(* CODESYS project timer.library
   Company: ESO
   Description: Local Device Control - Timer Library
   Version: 1.0.3.2
   Placeholder: ESO LDC Timer Library
   Author: Mario Kiekebusch
   Title: ESO LDC Timer Library

Project tree, tasks and I/O mapping:
  libraries: ESO MUDPI Library, * (ESO); Tc2_EtherCAT, * (Beckhoff Automation GmbH); Tc2_Standard, * (Beckhoff Automation GmbH); Tc2_System, * (Beckhoff Automation GmbH); Tc2_Utilities, * (Beckhoff Automation GmbH); Tc3_Module, * (Beckhoff Automation GmbH); VisuDialogs, * (System); VisuSymbols, 3.5.10.0 (System)
  DUTs/
    Enumerated/
      data type E_COE_PTP_ADDRESS_TYPE
      data type E_COE_PTP_DELAY_MECHANISM
      data type E_COE_PTP_STATE
      data type E_COE_PTP_TRANSPORT_LAYER
      data type E_COE_PTP_VERSION
      data type E_COE_STATE
      data type E_DIAG_STATE
      data type E_TIME_ERROR
      data type E_TIME_MODE
      data type E_TIME_SIGNAL_QOS
      data type E_TIME_SIGNAL_STATUS
      data type E_TIME_SOURCE
    Structures/
      data type T_COE_PTP_DIAGNOSTICS
      data type T_COE_PTP_ETHERNET
      data type T_COE_PTP_PARAMETERS
      data type T_COE_STAT
      data type T_DIAG_REP_CFG
      data type T_DIAG_REP_STAT
      data type T_IP_ADDRESS
      data type T_PAYLOAD
      data type T_TIME_CFG
      data type T_TIME_INFO
      data type T_TIME_SIGNAL
      data type T_TIME_STAT
  GVLs/
    global variables GVL_TimeConstants
  lib/
  POUs/
    function block FB_ReadEL6688CoE [ST]: DisableCoERead, ExecuteCoERead, FB_init, GetIpaAddr, GetLeapSecond, GetOffsetFromMaster, GetPtpState, IsErrorFree, ReadConfigParameters, ReadEthernetSettings, ReadLeapSecond, ReadOffsetFromMaster, ReadPtpState
    function block FB_SendEL6688Diag [ST]: FB_exit, FB_init, FB_reinit, IpAddressStringToInteger, ReceiveData, SendDiagnosticData, SetConfigurationParameters, TcAddRef, TcQueryInterface, TcRelease
    function block FB_TIME [ST]: CheckNtpSignal, CheckPtpSignal, ComputeNtpOffset, ComputePtpOffset, ComputeSimulationOffset, CycleUpdate, FB_init, GetErrorText, GetMode, GetMudpiTime, GetSource, GetTime, GetUtcTime, MudpiTimeToDc, PublishPtpDiagnostics, RPC_GetMode, RPC_GetUTC, RPC_SetMode, RPC_SetTime, SetDefaultMode, SetMode, SetSource, SetTime
    program MAIN [ST]
  Version/
    global variables Global_Version
  VISUs/
    Templates/
      visualisation GUI_TEMPLATE_TIME
    visualisation GUI_time_info
  text list GlobalTextList
*)

// DUTs/Enumerated/E_COE_PTP_ADDRESS_TYPE
{attribute 'qualified_only'}
{attribute 'strict'}
TYPE E_COE_PTP_ADDRESS_TYPE :
(
	UNKNOWN := -1,
	DHCP := 0,
	FIXED := 1
);
END_TYPE

// DUTs/Enumerated/E_COE_PTP_DELAY_MECHANISM
{attribute 'qualified_only'}
{attribute 'strict'}
TYPE E_COE_PTP_DELAY_MECHANISM :
(
	UNKNOWN := -1,
	DISABLED := 0,
	E2E := 1,
	P2P := 2
);
END_TYPE

// DUTs/Enumerated/E_COE_PTP_STATE
{attribute 'qualified_only'}
{attribute 'strict'}
TYPE E_COE_PTP_STATE :
(   
	UNKNOWN := -1,
	LISTENING := 4,
	SLAVE := 9
);
END_TYPE

// DUTs/Enumerated/E_COE_PTP_TRANSPORT_LAYER
{attribute 'qualified_only'}
{attribute 'strict'}
TYPE E_COE_PTP_TRANSPORT_LAYER :
(
	UNKNOWN := -1,
	PTP_OVER_ETHERNET := 0,
	PTP_OVER_UDP := 1
);
END_TYPE

// DUTs/Enumerated/E_COE_PTP_VERSION
{attribute 'qualified_only'}
{attribute 'strict'}
TYPE E_COE_PTP_VERSION :
(
	UNKONWN := -1,
	PTPv1 := 16,
	PTPv2 := 32
);
END_TYPE

// DUTs/Enumerated/E_COE_STATE
{attribute 'qualified_only'}
{attribute 'strict'}
TYPE E_COE_STATE :
(
	E_COE_UNKNOWN := -1,
	E_COE_NOT_STARTED := 0,	
	E_COE_INIT,
	E_COE_IDLE,
	E_COE_READ,
	E_COE_WAITING,
	E_COE_SLEEPING,
	E_COE_ERROR := 100
	
);
END_TYPE

// DUTs/Enumerated/E_DIAG_STATE
{attribute 'qualified_only'}
{attribute 'strict'}
TYPE E_DIAG_STATE :
(
	E_DIAG_DISABLED := -1,
	E_DIAG_INIT := 0,
	E_DIAG_SENDING,
	E_DIAG_WAITING
);
END_TYPE

// DUTs/Enumerated/E_TIME_ERROR
{attribute 'qualified_only'}
{attribute 'strict'}
TYPE E_TIME_ERROR :
(
	OK := 0,
	NO_SIMULATION_MODE,
	DC2TC_OFFSET_NOT_MAPPED,
	INT_EXT_NOT_MAPPED,
	COE_NOT_VALID,
	PTP_WRONG_STATE,
	PTP_NOT_SYNCHRONIZED,
	NTP_NOT_CONNECTED,
	NTP_NOT_SYNCHRONIZED
);
END_TYPE

// DUTs/Enumerated/E_TIME_MODE
{attribute 'qualified_only'}
{attribute 'strict'}
TYPE E_TIME_MODE :
(
	LOCAL,
    UTC_PTP,
	UTC_NTP,
	UTC,
    SIMULATION
);
END_TYPE

// DUTs/Enumerated/E_TIME_SIGNAL_QOS
{attribute 'qualified_only'}
{attribute 'strict'}
TYPE E_TIME_SIGNAL_QOS :
(
	NOT_VALID := 0,
	NOT_SYNCHRONIZED,
	VALID
);
END_TYPE

// DUTs/Enumerated/E_TIME_SIGNAL_STATUS
{attribute 'qualified_only'}
{attribute 'strict'}
TYPE E_TIME_SIGNAL_STATUS :
(
	CONNECTED := 0,
	NOT_CONNECTED
);
END_TYPE

// DUTs/Enumerated/E_TIME_SOURCE
{attribute 'qualified_only'}
{attribute 'strict'}
TYPE E_TIME_SOURCE :
(
	NONE,
	NTP,
    PTP
);
END_TYPE

// DUTs/Structures/T_COE_PTP_DIAGNOSTICS
TYPE T_COE_PTP_DIAGNOSTICS :
STRUCT
	ptp_state: E_COE_PTP_STATE := E_COE_PTP_STATE.UNKNOWN;
	leap_second: INT := 0;
	offset_from_master: DINT := 0;       // offset from master in ns
	offset_from_master_msec: LREAL := 0;  // offset from master in ms
	offset_from_master_sec: LREAL := 0;   // offset from master in sec
	mean_path_delay: DINT := 0;
END_STRUCT
END_TYPE

// DUTs/Structures/T_COE_PTP_ETHERNET
TYPE T_COE_PTP_ETHERNET :
STRUCT
	address_type: E_COE_PTP_ADDRESS_TYPE := E_COE_PTP_ADDRESS_TYPE.UNKNOWN;
	ip_address_arr:   DWORD;         
	ip_address:       T_IPv4Addr;
	subnet_mask_arr:  DWORD;
	subnet_mask:      T_IPv4Addr;
	gateway_arr:      DWORD;
	gateway:          T_IPv4Addr;
END_STRUCT
END_TYPE

// DUTs/Structures/T_COE_PTP_PARAMETERS
TYPE T_COE_PTP_PARAMETERS :
STRUCT
	ptp_version: E_COE_PTP_VERSION := E_COE_PTP_VERSION.UNKONWN;
	transport_layer: E_COE_PTP_TRANSPORT_LAYER := E_COE_PTP_TRANSPORT_LAYER.UNKNOWN;
	delay_mechanism : E_COE_PTP_DELAY_MECHANISM :=  E_COE_PTP_DELAY_MECHANISM.UNKNOWN;
	ethernet_settings: T_COE_PTP_ETHERNET;	
END_STRUCT
END_TYPE

// DUTs/Structures/T_COE_STAT
TYPE T_COE_STAT :
STRUCT
	diagnostics: T_COE_PTP_DIAGNOSTICS;
	config: T_COE_PTP_PARAMETERS;
	errorFlag: BOOL;
	errorNumber: UDINT;
END_STRUCT
END_TYPE

// DUTs/Structures/T_DIAG_REP_CFG
TYPE T_DIAG_REP_CFG :
STRUCT
	// Configuration parameters related to the TIME diagnostics.
	enabled : BOOL := FALSE; // True if diagnostic data is sent via MUDPI protocol
	address : Tc2_System.T_IPv4Addr := '134.171.2.213'; // Destination IP address for the data
	destination_port: UINT := 7003; // Destination port for the data
	source_port: UINT := 10000;    // Source port of the data
	topic_id: UDINT := 500;      // MUDPI Topic identity
	compontent_id: UINT := 1;  // MUDPI component identity
	sampling: UINT := 10000; // Sampling rate in milliseconds
END_STRUCT
END_TYPE

// DUTs/Structures/T_DIAG_REP_STAT
TYPE T_DIAG_REP_STAT :
STRUCT
	enabled: BOOL; // flag reporting if diagnostic data is being sent externally.
	state : E_DIAG_STATE := E_DIAG_STATE.E_DIAG_DISABLED;
	counter: UDINT; // counter the number of times the diagnostic data was sent.
	last_notification: LREAL; // timestamp of the last sent
	last_notification_date: STRING;
END_STRUCT
END_TYPE

// DUTs/Structures/T_IP_ADDRESS
TYPE T_IP_ADDRESS :
UNION
	ipAdrInternal : UDINT;
	ipAdr : ARRAY[0..3] OF BYTE;
END_UNION
END_TYPE

// DUTs/Structures/T_PAYLOAD
TYPE T_PAYLOAD :
STRUCT
	version:               UINT := 1;
	devtype:               UINT := 10;  // 10: is a Beckhoff PLC according ESO-331947
	hostname:              STRING(16) := '';
    port_state1:	       INT := 0;
	port_state2:           UINT := 0;
	offset_from_master:    LINT := 0;
	mean_path_delay:       ULINT := 0;
	announce_path_delay:   DINT := -1;
	sync_msg_count:        DINT := -1;
	delay_resp_count:      DINT := -1;
	clock_identity:        STRING(8) := '';
	gm_identity:           STRING(8) := '';
	parent_port_identity:  STRING(10) := '';
	current_utc_offset:    INT := 999;
	steps_removed:         UINT := 999;
	error_status:          UINT := 0;
	app_specific:          DINT := 0;
END_STRUCT
END_TYPE

// DUTs/Structures/T_TIME_CFG
TYPE T_TIME_CFG :
STRUCT
	nMode     : E_TIME_MODE := E_TIME_MODE.LOCAL;  // New mode configured.
	nSource   : E_TIME_SOURCE := E_TIME_SOURCE.NONE;  // New mode configured.
	sUserTime : STRING(29) := 'YYYY-MM-DD-hh:mm:ss.nnnnnnnnn'; // Last user configured datetime in format YYYY-MM-DD-hh:mm:ss.nnnnnnnnn
	tUserTime : ULINT := 0;
	nLeapSecond: INT := 37; // Leap second to convert to TAI for systems without PTP.
	
    diag_report: T_DIAG_REP_CFG;	
END_STRUCT
END_TYPE

// DUTs/Structures/T_TIME_INFO
TYPE T_TIME_INFO :
STRUCT
	time_offset :    LINT;
	leap_second:    DINT;  
	time_mode   :    DINT := E_TIME_MODE.LOCAL;
END_STRUCT
END_TYPE

// DUTs/Structures/T_TIME_SIGNAL
TYPE T_TIME_SIGNAL :
STRUCT
	status : E_TIME_SIGNAL_STATUS := E_TIME_SIGNAL_STATUS.NOT_CONNECTED;
	qos    : E_TIME_SIGNAL_QOS    := E_TIME_SIGNAL_QOS.NOT_VALID;
	time_difference : UDINT; // Time difference between DC and External Time Source
	
END_STRUCT
END_TYPE

// DUTs/Structures/T_TIME_STAT
TYPE T_TIME_STAT :
STRUCT
	sLibVersion:	   STRING	:= 'UNKNOWN'; // Library version as string, e.g. '1.2.0.0'
	sSystemTime:       STRING := '';
	sDcTime:           STRING := '';
	sUtcTime:          STRING := '';
	sTaiTime:          STRING := '';
	sErrorMsg:         STRING := '';
	mode:              E_TIME_MODE := E_TIME_MODE.LOCAL;
	source:			   E_TIME_SOURCE := E_TIME_SOURCE.NTP;
	signal:            T_TIME_SIGNAL;
	lNtpOffsetTime:    LINT := 0;
	lPtpOffsetTime:    LINT := 0;
	lSimOffsetTime:    LINT := 0;
	lDcCurrentTime:    LINT := 0;
	lUtcTime:          LINT := 0;   // UTC time in nanoseconds
	lTaiTime:          LINT := 0;   // TAI time in nanoseconds 
	lTaiUnixTime:      LINT := 0;   // UNIX time in nanoseconds
	lrTaiUnixTimeinSecs: LREAL := 0; // UNIX time in seconds - used in MUDPI protocol
	
	sUserTime:         STRING(29) := 'YYYY-MM-DD-hh:mm:ss.nnnnnnnnn'; // Last user configured datetime in format YYYY-MM-DD-hh:mm:ss.nnnnnnnnn
	tUserTime :        ULINT := 0;
	el6688:            T_COE_STAT; 
	diag_report:       T_DIAG_REP_STAT;
	
END_STRUCT
END_TYPE

// GVLs/GVL_TimeConstants
{attribute 'qualified_only'}
VAR_GLOBAL
	C_INVALID:    DINT := -9999;
	C_ONE_SEC:    LINT := 1000000000;
	C_STAT_OK:    DINT := 0;
	C_NS2MSEC:    LREAL := 1/1E+6;
	C_NS2SEC:     LREAL := 1/1E+9;
	C_UNIX_OFFSET_SEC: ULINT := DATE_TO_ULINT(DATE#2000-01-01); // 946,684,800 seconds = 15,778,080 minutes = 262,968 hours
	C_UNIX_OFFSET_MICROSEC:  ULINT := C_UNIX_OFFSET_SEC * 10#1000_000;
END_VAR

// Version/Global_Version
{attribute 'TcGenerated'}
{attribute 'no-analysis'}
{attribute 'linkalways'}
// This function has been automatically generated from the project information.
VAR_GLOBAL CONSTANT
	{attribute 'const_non_replaced'}
	stLibVersion_ESO_LDC_Timer_Library : ST_LibVersion := (iMajor := 1, iMinor := 0, iBuild := 3, iRevision := 2, nFlags := 0, sVersion := '1.0.3.2');
END_VAR

// POUs/FB_ReadEL6688CoE
FUNCTION_BLOCK FB_ReadEL6688CoE
VAR_INPUT
	st_amsAddr:  AMSADDR;
END_VAR
VAR_OUTPUT
END_VAR


VAR_IN_OUT
	i_coe_stat               : T_COE_STAT;
END_VAR

VAR
	  stat: REFERENCE TO T_COE_STAT;
	        
	  fb_SdoLeapSecond   : FB_EcCoESdoRead;
	  fb_SdoPtpState     : FB_EcCoESdoRead;
	  fb_SdoOffset       : FB_EcCoESdoRead;
	  
	  fb_SdoDelayMech    : FB_EcCoESdoRead;
	  fb_SdoPtpVersion   : FB_EcCoESdoRead;
	  fb_SdoTransLayer   : FB_EcCoESdoRead;
	  
	  fb_SdoEtherType    : FB_EcCoESdoRead;
	  fb_SdoEtherIp      : FB_EcCoESdoRead;
	  fb_SdoEtherMask    : FB_EcCoESdoRead;
	  fb_SdoEtherGateway : FB_EcCoESdoRead;
	  
	  
      s_mNetId           : T_AmsNetId;
      b_mCoEExecute      : BOOL;
      n_mSlaveAddr       : UINT;
	  b_CoEReadDiag      : BOOL;    // Flag to trigger reading of diagnostics CoE parameters
	  b_CoEReadCfg       : BOOL;    // Flag to trigger reading of configuration CoE parameters
	  n_state            : E_COE_STATE := E_COE_STATE.E_COE_UNKNOWN;
	  
	  waitTime			 : TIME := T#10000MS;
	  initTime			 : TIME := T#5MS;
	  waitTout			 : TON;    // timer for resting time when reading CoE parameters.
      initTout			 : TON;    // timer for waiting few ms before start reading CoE
END_VAR

stat REF= i_coe_stat; 

CASE n_state OF
	E_COE_STATE.E_COE_NOT_STARTED:
	    initTout (IN := TRUE, PT := initTime); (* enable timer *)
		n_state := E_COE_STATE.E_COE_INIT;
		
	E_COE_STATE.E_COE_INIT:
	    initTout (IN := TRUE);  (* activate timer counting per each cycle *)
		IF initTout.Q THEN
	       n_state := E_COE_STATE.E_COE_IDLE;
		   s_mNetId := F_CreateAmsNetId(st_amsAddr.netId);
		   n_mSlaveAddr := st_amsAddr.port;
		   b_CoEReadCfg := TRUE;
		   b_CoEReadDiag := TRUE;
		   initTout (IN := FALSE);
		END_IF
		
	E_COE_STATE.E_COE_IDLE:
	    waitTout (IN := FALSE); (* Reset timer *)
		DisableCoERead();
	
		 IF (b_CoEReadCfg OR b_CoEReadDiag) THEN
			// Prepare CoE-Access: Read value of CoE object/ sub index
			n_state := E_COE_STATE.E_COE_READ;// Next state for writing
		END_IF
	   
		
	E_COE_STATE.E_COE_READ:
	    waitTout (IN := FALSE); (* Reset timer *)
		stat.errorFlag := FALSE;
	   	stat.errorNumber := 0;
		IF (b_CoEReadCfg) THEN
		 	ReadConfigParameters(st_ioParams := stat.config);	
			b_CoEReadCfg := FALSE;
		END_IF
		IF (b_CoEReadDiag) THEN
	    	ReadLeapSecond(n_iIndex := 16#FA80, 
				n_iSubindex := 11, 
				n_ioLeapSecond := stat.diagnostics.leap_second);
			ReadPtpState(n_iIndex := 16#FA80, 
				n_iSubindex := 2, 
				n_ioPtpState := stat.diagnostics.ptp_state);
	    	ReadOffsetFromMaster(n_iIndex := 16#FA80, 
				n_iSubindex := 6, 
				n_ioOffsetFromMaster := stat.diagnostics.offset_from_master);
			b_CoEReadDiag := FALSE;
		END_IF
				
		n_state := E_COE_STATE.E_COE_WAITING;
		
	E_COE_STATE.E_COE_WAITING:
	    // Execute CoE read until done
				
		ExecuteCoERead(fb_SdoPtpVersion);
		ExecuteCoERead(fb_SdoDelayMech);
		ExecuteCoERead(fb_SdoTransLayer);
	    ExecuteCoERead(fb_SdoEtherType);
		ExecuteCoERead(fb_SdoEtherIp);
		ExecuteCoERead(fb_SdoEtherMask);
		ExecuteCoERead(fb_SdoEtherGateway);
		
	    ExecuteCoERead(fb_SdoLeapSecond);  
		ExecuteCoERead(fb_SdoPtpState);
		ExecuteCoERead(fb_SdoOffset);
			
		IF (NOT fb_SdoEtherType.bBusy) AND
			(NOT fb_SdoEtherIp.bBusy) AND
			(NOT fb_SdoEtherMask.bBusy) AND
			(NOT fb_SdoEtherGateway.bBusy) AND
			(NOT fb_SdoDelayMech.bBusy) AND
			(NOT fb_SdoTransLayer.bBusy) AND
			(NOT fb_SdoPtpVersion.bBusy) AND
			(NOT fb_SdoLeapSecond.bBusy) AND
			(NOT fb_SdoPtpState.bBusy) AND
			(NOT fb_SdoOffset.bBusy) THEN
			    stat.config.ethernet_settings.ip_address := GetIpaAddr(stat.config.ethernet_settings.ip_address_arr);
				stat.config.ethernet_settings.subnet_mask := GetIpaAddr(stat.config.ethernet_settings.subnet_mask_arr);
				stat.config.ethernet_settings.gateway := GetIpaAddr(stat.config.ethernet_settings.gateway_arr);
				stat.diagnostics.offset_from_master_msec := DINT_TO_LREAL(stat.diagnostics.offset_from_master) * GVL_TimeConstants.C_NS2MSEC;
				stat.diagnostics.offset_from_master_sec := DINT_TO_LREAL(stat.diagnostics.offset_from_master) * GVL_TimeConstants.C_NS2SEC;
				n_state := E_COE_STATE.E_COE_SLEEPING;
		END_IF
			
	
		waitTout (IN := TRUE, PT := waitTime); (* enable timer *)
		
	E_COE_STATE.E_COE_SLEEPING:
		DisableCoERead();
	   
		waitTout (IN := TRUE);  (* activate timer counting per each cycle *)
		IF waitTout.Q THEN
	       n_state := E_COE_STATE.E_COE_IDLE;
		   b_CoEReadDiag := TRUE;
		   waitTout (IN := FALSE);
		END_IF
		
	E_COE_STATE.E_COE_ERROR:
       waitTout (IN := FALSE);	
	   waitTout (IN := TRUE, PT := waitTime); (* enable timer *)
	   // TODO: Log the error
	   n_state := E_COE_STATE.E_COE_SLEEPING;
END_CASE

METHOD DisableCoERead
VAR_INPUT
END_VAR

 // CoE configuration parameters
 fb_SdoPtpVersion(bExecute:=FALSE);
 fb_SdoDelayMech(bExecute:=FALSE);
 fb_SdoTransLayer(bExecute:=FALSE);
 fb_SdoEtherType(bExecute:=FALSE);
 fb_SdoEtherIp(bExecute:=FALSE);
 fb_SdoEtherMask(bExecute:=FALSE);
 fb_SdoEtherGateway(bExecute:=FALSE);
	
 // CoE diagnostic parameters
 fb_SdoLeapSecond(bExecute:=FALSE);
 fb_SdoPtpState(bExecute:=FALSE);
 fb_SdoOffset(bExecute:=FALSE);
END_METHOD

METHOD ExecuteCoERead : BOOL

VAR_IN_OUT
	refFb :FB_EcCoESdoRead;
END_VAR

refFb();

IF refFb.bError THEN
	stat.errorFlag := refFb.bError;
	stat.errorNumber := refFb.nErrId;
	n_state := E_COE_STATE.E_COE_ERROR;
END_IF
END_METHOD

METHOD FB_init : BOOL
VAR_INPUT
	bInitRetains : BOOL; // if TRUE, the retain variables are initialized (warm start / cold start)
	bInCopyCode : BOOL;  // if TRUE, the instance afterwards gets moved into the copy code (online change)
END_VAR

initTout (IN := FALSE); (* Reset timer *)
n_state := E_COE_STATE.E_COE_NOT_STARTED;
END_METHOD

METHOD GetIpaAddr : T_IPv4Addr
VAR_INPUT
	in_word : DWORD;
END_VAR

VAR
  ids     : T_IPv4AddrArr := [0, 0, 0, 0];  
  bo_word : DWORD := 0;	
  sIPv4   : T_IPv4Addr := '';
END_VAR

// values in terminal EL6688 have network byte order.
bo_word := BE32_TO_HOST(in_word);

// In order to conver to string using system function, we need an array of bytes.
memcpy(ADR(ids), ADR(bo_word), SIZEOF(bo_word));
	
sIPv4 := F_CreateIPv4Addr( ids );

GetIpaAddr := sIPv4;
RETURN;
END_METHOD

METHOD GetLeapSecond : INT
VAR_INPUT
END_VAR

GetLeapSecond := stat.diagnostics.leap_second;
END_METHOD

METHOD GetOffsetFromMaster : DINT
VAR_INPUT
END_VAR

GetOffsetFromMaster := stat.diagnostics.offset_from_master;
END_METHOD

METHOD GetPtpState : INT
VAR_INPUT
END_VAR
GetPtpState := stat.diagnostics.ptp_state;
END_METHOD

METHOD IsErrorFree : BOOL
VAR_INPUT
END_VAR

IF NOT stat.errorFlag THEN
	IsErrorFree := TRUE;
	return;
END_IF

IsErrorFree := FALSE;
END_METHOD

METHOD ReadConfigParameters 
VAR_INPUT
END_VAR

VAR_IN_OUT
	st_ioParams : T_COE_PTP_PARAMETERS;
END_VAR

fb_SdoPtpVersion(sNetId:= s_mNetId,
    nSlaveAddr := n_mSlaveAddr,
	nIndex := 16#F880, 
	nSubIndex := 1, 
	pDstBuf := ADR(st_ioParams.ptp_version), 
	cbBufLen := SIZEOF(st_ioParams.ptp_version),
	bExecute := TRUE);
	
fb_SdoTransLayer(sNetId:= s_mNetId,
    nSlaveAddr := n_mSlaveAddr,
	nIndex := 16#F882, 
	nSubIndex := 1, 
	pDstBuf := ADR(st_ioParams.transport_layer), 
	cbBufLen := SIZEOF(st_ioParams.transport_layer),
	bExecute := TRUE);
	
 fb_SdoDelayMech(sNetId:= s_mNetId,
    nSlaveAddr := n_mSlaveAddr,
	nIndex := 16#F882, 
	nSubIndex := 5, 
	pDstBuf := ADR(st_ioParams.delay_mechanism), 
	cbBufLen := SIZEOF(st_ioParams.delay_mechanism),
	bExecute := TRUE);

ReadEthernetSettings(n_iIndex := 16#F8E0, 
				st_ioEthernetSettings := st_ioParams.ethernet_settings);
END_METHOD

METHOD ReadEthernetSettings
VAR_INPUT
	n_iIndex     : WORD ;
END_VAR

VAR_IN_OUT
	st_ioEthernetSettings : T_COE_PTP_ETHERNET;
END_VAR

VAR 

END_VAR


fb_SdoEtherType(sNetId:= s_mNetId,
    nSlaveAddr := n_mSlaveAddr,
	nIndex := n_iIndex, 
	nSubIndex := 1, 
	pDstBuf := ADR(st_ioEthernetSettings.address_type), 
	cbBufLen := SIZEOF(st_ioEthernetSettings.address_type),
	bExecute := TRUE);
	
fb_SdoEtherIp(sNetId:= s_mNetId,
    nSlaveAddr := n_mSlaveAddr,
	nIndex := n_iIndex, 
	nSubIndex := 2, 
	pDstBuf := ADR(st_ioEthernetSettings.ip_address_arr), 
	cbBufLen := SIZEOF(st_ioEthernetSettings.ip_address_arr),
	bExecute := TRUE);

	
	
	
fb_SdoEtherMask(sNetId:= s_mNetId,
    nSlaveAddr := n_mSlaveAddr,
	nIndex := n_iIndex, 
	nSubIndex := 3, 
	pDstBuf := ADR(st_ioEthernetSettings.subnet_mask_arr), 
	cbBufLen := SIZEOF(st_ioEthernetSettings.subnet_mask_arr),
	bExecute := TRUE);
	
	
	
fb_SdoEtherGateway(sNetId:= s_mNetId,
    nSlaveAddr := n_mSlaveAddr,
	nIndex := n_iIndex, 
	nSubIndex := 4, 
	pDstBuf := ADR(st_ioEthernetSettings.gateway_arr), 
	cbBufLen := SIZEOF(st_ioEthernetSettings.gateway_arr),
	bExecute := TRUE);
END_METHOD

METHOD ReadLeapSecond : BOOL
VAR_INPUT
	n_iIndex     : WORD ;
	n_iSubindex  : BYTE;
END_VAR

VAR_IN_OUT
	n_ioLeapSecond : INT;
END_VAR
		
//IF (b_CoERead = TRUE) THEN
fb_SdoLeapSecond(sNetId:= s_mNetId,
    nSlaveAddr := n_mSlaveAddr,
	nIndex := n_iIndex, 
	nSubIndex := n_iSubindex, 
	pDstBuf := ADR(n_ioLeapSecond), 
	cbBufLen := SIZEOF(n_ioLeapSecond),
	bExecute := TRUE);
								  
(* Prevent reading more than once the parameter *)			
//b_CoERead := FALSE;
END_METHOD

METHOD ReadOffsetFromMaster : BOOL
VAR_INPUT
	n_iIndex     : WORD ;
	n_iSubindex  : BYTE;
END_VAR

VAR_IN_OUT
	n_ioOffsetFromMaster : DINT;
END_VAR

fb_SdoOffset(sNetId:= s_mNetId,
    nSlaveAddr := n_mSlaveAddr,
	nIndex := n_iIndex, 
	nSubIndex := n_iSubindex, 
	pDstBuf := ADR(n_ioOffsetFromMaster), 
	cbBufLen := SIZEOF(n_ioOffsetFromMaster),
	bExecute := TRUE);
END_METHOD

METHOD ReadPtpState : BOOL
VAR_INPUT
	n_iIndex     : WORD ;
	n_iSubindex  : BYTE;
END_VAR

VAR_IN_OUT
	n_ioPtpState : INT;
END_VAR

fb_SdoPtpState(sNetId:= s_mNetId,
    nSlaveAddr := n_mSlaveAddr,
	nIndex := n_iIndex, 
	nSubIndex := n_iSubindex, 
	pDstBuf := ADR(n_ioPtpState), 
	cbBufLen := SIZEOF(n_ioPtpState),
	bExecute := TRUE);
END_METHOD

END_FUNCTION_BLOCK

// POUs/FB_SendEL6688Diag
(*
    This function blocks aims to pack the EL6688 diagnostic data in MUDPI frames
    and transmit them to Time System using Beckhoffs realtime UDP driver (TF6311). 
    The user of this function blocks needs to do the following in order for the library to work correctly:
    - Initialize the library with configuration parameters
        - Destination IP-address (a multicast address)
        - Destination port
        - Source port
        - Topic identity (see MUDPI-specification)
        - Component identity (see MUDPI-specification)
*)

{attribute 'c++_compatible'}
FUNCTION_BLOCK FB_SendEL6688Diag IMPLEMENTS ITcIoUdpProtocolRecv
VAR_INPUT
END_VAR
VAR_OUTPUT
END_VAR
VAR
	(* TF6311 realtime driver parameters *)
    {attribute 'TcInitSymbol'}
    oid : OTCID;
    ipUdp : ITcIoUdpProtocol;
	nUdpPort : UINT := 10000;
    nReceivedPackets : UINT;
    uLastReceivedIP : T_IP_ADDRESS;
    hrInit : HRESULT;
    hrSend : HRESULT; 
    bSuccessfulInitializationOfRealtimeDriver : BOOL := FALSE; // Indication of whether the realtime driver is properly initialized.

	(* Data/contents parameters *)
    mudpiPacket : ESO_MUDPI.FB_MudpiPacket(topicId := 500, componentId := 10);
    dataToBeSent : ARRAY[0..23] OF BYTE; // 6 parameters, each 4 bytes = 24 bytes
	
	  (* Transmission/communication parameters *)
    _destinationIpAddress : UDINT; // Destination address for the data
    _destinationPort : UINT; // Destination port for the data
    _sourcePort : UINT; // Source port of the data
	
END_VAR

METHOD FB_exit : BOOL
VAR_INPUT
    bInCopyCode : BOOL; // if TRUE, the exit method is called for exiting an instance that is copied afterwards (online change).
END_VAR
IF NOT bInCopyCode THEN // no online change
    IF ipUdp <> 0 THEN
        //ipUdp.UnregisterReceiver(nUdpPort); // Shutdown
        ipUdp.UnregisterReceiver(nUdpPort); // Shutdown
        FW_SafeRelease(ADR(ipUdp));
        FB_exit := TRUE;
    END_IF
END_IF
END_METHOD

METHOD FB_init : BOOL
VAR_INPUT
    bInitRetains : BOOL; // if TRUE, the retain variables are initialized (warm start / cold start)
    bInCopyCode : BOOL;  // if TRUE, the instance afterwards gets moved into the copy code (online change)
END_VAR
MudpiPacket.SetNumFrames(NumFrames := 1);
MudpiPacket.SetFrameId(FrameId := 1);

(*
IF NOT bInCopyCode THEN // no online change
	IF ipUdp = 0 AND oid <> 0 THEN
	    hrInit := FW_ObjMgr_GetObjectInstance(	oid:=oid, 
											iid:=TC_GLOBAL_IID_LIST.IID_ITcIoUdpProtocol, 
											pipUnk:=ADR(ipUdp) );
		IF SUCCEEDED(hrInit) THEN 
			IF  SUCCEEDED(ipUdp.RegisterReceiver(nUdpPort, THIS^)) THEN //open port
				FB_init := TRUE;
			ELSE 
				FB_init := FALSE; 
				FW_SafeRelease(ADR(ipUdp));
			END_IF
		END_IF
	ELSIF oid = 0 THEN 
		FB_init := FALSE; 
		hrInit := ERR_INVALID_PARAM; 				
	END_IF
END_IF
*)
END_METHOD

METHOD FB_reinit : BOOL
IF (ipUdp <> 0) THEN
    //ipUdp.RegisterReceiver(nUdpPort, THIS^);
    ipUdp.RegisterReceiver(nUdpPort, THIS^);
    FB_reinit := TRUE;
END_IF
END_METHOD

METHOD PRIVATE IpAddressStringToInteger : UDINT
VAR_INPUT
    IpAddress : Tc2_System.T_IPv4Addr;
END_VAR
VAR
    IpAddressArray : Tc2_System.T_IPv4AddrArr;
    IpAddressInteger : UDINT;
END_VAR
IpAddressArray := Tc2_System.F_ScanIPv4AddrIds(sIPv4 := IpAddress);
IpAddressInteger := LREAL_TO_UDINT(IpAddressArray[0] * EXPT(256, 3) +
                                   IpAddressArray[1] * EXPT(256, 2) +
                                   IpAddressArray[2] * EXPT(256, 1) +
                                   IpAddressArray[3]);

IpAddressStringToInteger := IpAddressInteger;
END_METHOD

{attribute 'c++_compatible'}
{attribute 'minimal_input_size' := '4'}
{attribute 'pack_mode' := '4'}
{warning 'add method implementation'}
METHOD ReceiveData : HRESULT
VAR_INPUT
	ipAddr	: UDINT;
	udpDestPort	: UINT;
	udpSrcPort	: UINT;
	nData	: UDINT;
	pData	: PVOID;
	pVlan	: POINTER TO ETYPE_VLAN_HEADER := 0;
END_VAR
nReceivedPackets := nReceivedPackets + 1;
uLastReceivedIP.ipAdrInternal := ipAddr;
END_METHOD

(*
    This method carry out the sending of the diagnostic data using the Ethernet network driver.
    The parameters are the array of data to be sent and the timestamp that is required by
	the MUDPI protocol.
*)

METHOD SendDiagnosticData : HRESULT
VAR_INPUT
	payload : POINTER TO T_PAYLOAD; 
	timeStamp : LREAL;
END_VAR
	
VAR
	dataToBeSent : ARRAY[0..87] OF BYTE; 
	
END_VAR


IF ipUdp <> 0 AND bSuccessfulInitializationOfRealtimeDriver = TRUE THEN
	
    // Fill up vector with structure
	memcpy(ADR(dataToBeSent[0]),  ADR(payload^.version), SIZEOF(payload^.version));
	memcpy(ADR(dataToBeSent[2]),  ADR(payload^.devtype), SIZEOF(payload^.devtype));
	memcpy(ADR(dataToBeSent[4]),  ADR(payload^.hostname), SIZEOF(payload^.hostname));
	memcpy(ADR(dataToBeSent[20]), ADR(payload^.port_state1), SIZEOF(payload^.port_state1));
	memcpy(ADR(dataToBeSent[22]), ADR(payload^.port_state2), SIZEOF(payload^.port_state2));
	memcpy(ADR(dataToBeSent[24]), ADR(payload^.offset_from_master), SIZEOF(payload^.offset_from_master));
	memcpy(ADR(dataToBeSent[32]), ADR(payload^.mean_path_delay), SIZEOF(payload^.mean_path_delay));
	memcpy(ADR(dataToBeSent[40]), ADR(payload^.announce_path_delay), SIZEOF(payload^.announce_path_delay));
	memcpy(ADR(dataToBeSent[44]), ADR(payload^.sync_msg_count), SIZEOF(payload^.sync_msg_count));
	memcpy(ADR(dataToBeSent[48]), ADR(payload^.delay_resp_count), SIZEOF(payload^.delay_resp_count));
	memcpy(ADR(dataToBeSent[52]), ADR(payload^.clock_identity), SIZEOF(payload^.clock_identity));
	memcpy(ADR(dataToBeSent[60]), ADR(payload^.gm_identity), SIZEOF(payload^.gm_identity));
	memcpy(ADR(dataToBeSent[68]), ADR(payload^.parent_port_identity), SIZEOF(payload^.parent_port_identity));
	memcpy(ADR(dataToBeSent[78]), ADR(payload^.current_utc_offset), SIZEOF(payload^.current_utc_offset));
	memcpy(ADR(dataToBeSent[80]), ADR(payload^.steps_removed), SIZEOF(payload^.steps_removed));
	memcpy(ADR(dataToBeSent[82]), ADR(payload^.error_status), SIZEOF(payload^.error_status));
	memcpy(ADR(dataToBeSent[84]), ADR(payload^.app_specific), SIZEOF(payload^.app_specific));
	
    // Build MUDPI packet
	mudpiPacket.SetTimeStamp(Timestamp := timeStamp);
    mudpiPacket.SetPayload(payload := ADR(dataToBeSent),
                           payloadSize := SIZEOF(dataToBeSent));
						   
	// Send Data via UDP
    hrSend := ipUdp.SendData(ipDestAddr := _DestinationIpAddress,
                             udpDestPort := _DestinationPort,
                             udpSrcPort := _SourcePort,
                             nData := mudpiPacket.Size(),
                             pData := mudpiPacket.Data(),
                             bCalcUdpCheckSum := FALSE,
                             pVlan := 0);
    IF SUCCEEDED(hrSend) THEN
        mudpiPacket.IncreaseSampleId();
	END_IF
END_IF
END_METHOD

METHOD PUBLIC SetConfigurationParameters
VAR_INPUT
    DestinationIpAddress : Tc2_System.T_IPv4Addr; // Destination IP address for the data
    DestinationPort : UINT; // Destination port for the data
    SourcePort : UINT; // Source port of the data
    TopicId : UDINT; // MUDPI Topic identity
    ComponentId : UINT; // MUDPI component identity
END_VAR
mudpiPacket.SetTopicId(TopicId := TopicId);
mudpiPacket.SetComponentId(ComponentId := ComponentId);

_DestinationIpAddress := IpAddressStringToInteger(IpAddress := DestinationIpAddress);
_DestinationPort := DestinationPort;
_SourcePort := SourcePort;

IF ipUdp = 0 AND NOT bSuccessfulInitializationOfRealtimeDriver THEN
    hrInit := FW_ObjMgr_GetObjectInstance(oid := oid, 
                                          iid := TC_GLOBAL_IID_LIST.IID_ITcIoUdpProtocol,
                                          pipUnk := ADR(ipUdp));
    IF SUCCEEDED(hrInit) THEN
        IF SUCCEEDED(ipUdp.RegisterReceiver(_SourcePort, THIS^)) THEN //open port
            bSuccessfulInitializationOfRealtimeDriver := TRUE;
        ELSE
            FW_SafeRelease(ADR(ipUdp));
        END_IF
    END_IF
END_IF
END_METHOD

{attribute 'c++_compatible'}
{attribute 'minimal_input_size' := '4'}
{attribute 'pack_mode' := '4'}
{warning 'add method implementation'}
METHOD TcAddRef : UDINT
END_METHOD

{attribute 'object_name' := 'TcQueryInterface'}
{attribute 'c++_compatible'}
{attribute 'signature_flag' := '33554688'}
{attribute 'pack_mode' := '4'}
{attribute 'show'}
{attribute 'minimal_input_size' := '4'}
METHOD TcQueryInterface : HRESULT
VAR_INPUT
	iid	: REFERENCE TO IID;
	pipItf	: POINTER TO PVOID;
END_VAR
VAR
	ipUdpRecv : ITcIoUdpProtocolRecv;
	ipUnknown : ITcUnknown;	
END_VAR
IF GuidsEqual(ADR(iid), ADR(TC_GLOBAL_IID_LIST.IID_ITcIoUdpProtocolRecv)) THEN
	ipUdpRecv := THIS^; // cast to interface pointer
	pipItf^ := ITCUNKNOWN_TO_PVOID(ipUdpRecv);
	TcAddRef();
	TcQueryInterface := S_OK;
ELSIF GuidsEqual(ADR(iid), ADR(TC_GLOBAL_IID_LIST.IID_ITcUnknown)) THEN
	ipUnknown := THIS^; // cast to interface pointer
	pipItf^ := ITCUNKNOWN_TO_PVOID(ipUnknown);
	TcAddRef();
	TcQueryInterface := S_OK;
ELSE
	TcQueryInterface := E_HRESULTAdsErr.NOINTERFACE ; //Call super if this fb extends some other
END_IF
END_METHOD

{attribute 'c++_compatible'}
{attribute 'minimal_input_size' := '4'}
{attribute 'pack_mode' := '4'}
{warning 'add method implementation'}
METHOD TcRelease : UDINT
END_METHOD

END_FUNCTION_BLOCK

// POUs/FB_TIME
FUNCTION_BLOCK FB_TIME
VAR_INPUT
END_VAR
VAR_OUTPUT
END_VAR
VAR
	{attribute 'OPC.UA.DA' := '1'}
	{attribute 'OPC.UA.DA.Access' := '1'}
	stat:		T_TIME_STAT;

	{attribute 'OPC.UA.DA' := '1'}
    cfg:         T_TIME_CFG;	
	
	{attribute 'OPC.UA.DA' := '0'}
	fb_CoE:         FB_ReadEL6688CoE;
	
	{attribute 'OPC.UA.DA' := '0'}
	fb_SendDiag:         FB_SendEL6688Diag;
	
	// Input variables from EL6688 
	{attribute 'OPC.UA.DA' := '0'}
	i_inTime               AT %I* : ULINT := 0;
	{attribute 'OPC.UA.DA' := '0'}
	i_exTime               AT %I* : ULINT := 0;
	{attribute 'OPC.UA.DA' := '0'}
	i_dc2TcOffset          AT %I* : LINT := GVL_TimeConstants.C_INVALID;
	{attribute 'OPC.UA.DA' := '0'}
	i_dc2ExtOffset         AT %I* : LINT := GVL_TimeConstants.C_INVALID;
	{attribute 'OPC.UA.DA' := '0'}
	i_extDevNotConnected   AT %I* : BOOL := TRUE;
	{attribute 'OPC.UA.DA' := '0'}
	i_syncMode             AT %I* : UINT;
	{attribute 'OPC.UA.DA' := '0'}
	i_AdsAddr	           AT %I*:	AMSADDR;				// ADS address structure
	{attribute 'OPC.UA.DA' := '0'}
	
	// Input variables from NTP
	{attribute 'OPC.UA.DA' := '0'}
    i_exNtpExtTime               AT %I* : LINT := 0;
	
	{attribute 'OPC.UA.DA' := '0'}
    i_exNtpSysTime         AT %I* : LINT := 0;
	
	{attribute 'OPC.UA.DA' := '0'}
    i_exNtpExtOffset         AT %I* : LINT := 0;
	
	{attribute 'OPC.UA.DA' := '0'}
	i_exNtpConnected   AT %I* : BOOL := FALSE;
	
	{attribute 'OPC.UA.DA' := '0'}
	i_exNtpSynchronized  AT %I* : BOOL := FALSE;
	
	
 	{attribute 'OPC.UA.DA' := '0'}
	q_timeInfo             AT %Q*: T_TIME_INFO;    
	
	rtrigEnableDiagReport        : R_TRIG;
    ftrigDisableDiagReport       : F_TRIG;  
	waitTime			 : TIME := T#10000MS;
	waitTout			 : TON;    // timer for resting time when reading CoE parameters.
	payload              : T_PAYLOAD;
	   
	
END_VAR


fb_CoE(st_amsAddr := i_AdsAddr, i_coe_stat := stat.el6688);
fb_SendDiag();

CycleUpdate();

// If TIMER is configured to send diagnostic reports to the Time System then
// it enables the sending of the data.
rtrigEnableDiagReport(CLK := cfg.diag_report.enabled);
ftrigDisableDiagReport(CLK := cfg.diag_report.enabled);

// Check for the rising edge of the enable flag
IF rtrigEnableDiagReport.Q THEN
	stat.diag_report.state := E_DIAG_STATE.E_DIAG_INIT;
	stat.diag_report.enabled := TRUE;
END_IF

// Check for the falling edge of the enable flag
IF ftrigDisableDiagReport.Q THEN
	stat.diag_report.state := E_DIAG_STATE.E_DIAG_DISABLED;
	stat.diag_report.counter := 0;
	stat.diag_report.enabled := FALSE;
END_IF

CASE stat.diag_report.state OF
E_DIAG_STATE.E_DIAG_INIT:

	fb_SendDiag.SetConfigurationParameters(DestinationIpAddress := cfg.diag_report.address,
		DestinationPort := cfg.diag_report.destination_port,
		SourcePort := cfg.diag_report.source_port,
		TopicId := cfg.diag_report.topic_id,
		ComponentId := cfg.diag_report.compontent_id);
	
	IF DINT_TO_TIME(cfg.diag_report.sampling) < T#500MS THEN
		waitTime := T#500MS;
	ELSE
		waitTime :=  DINT_TO_TIME(cfg.diag_report.sampling);
	END_IF	
	waitTout (IN := TRUE, PT := waitTime); (* enable timer *)
	
	stat.diag_report.state := E_DIAG_STATE.E_DIAG_WAITING;
E_DIAG_STATE.E_DIAG_WAITING:	
	waitTout (IN := TRUE);  (* activate timer counting per each cycle *)
 	IF waitTout.Q THEN
		waitTout (IN := FALSE);
		stat.diag_report.state := E_DIAG_STATE.E_DIAG_SENDING;
 	END_IF
E_DIAG_STATE.E_DIAG_SENDING:  
	// Added information to the payload structure
	// Not all fields are currently supported.
 	payload.port_state1 := fb_CoE.GetPtpState();
	payload.offset_from_master := fb_CoE.GetOffsetFromMaster();
	payload.current_utc_offset := fb_CoE.GetLeapSecond();
	
    fb_SendDiag.SendDiagnosticData(payload := ADR(payload),
					timeStamp := stat.lrTaiUnixTimeinSecs) ;	
	stat.diag_report.counter := stat.diag_report.counter + 1;
	// Reset timer
	waitTout (IN := FALSE);  
	// Go back to the init
	stat.diag_report.state := E_DIAG_STATE.E_DIAG_INIT;
END_CASE

METHOD CheckNtpSignal : BOOL
VAR_INPUT
END_VAR
stat.signal.status :=  E_TIME_SIGNAL_STATUS.CONNECTED;
stat.signal.qos := E_TIME_SIGNAL_QOS.VALID;


// Check external signal. This variable must be mapped to the EL6688 terminal.
IF (NOT i_exNtpConnected) THEN
	stat.signal.status :=  E_TIME_SIGNAL_STATUS.NOT_CONNECTED;
	stat.signal.qos := E_TIME_SIGNAL_QOS.NOT_VALID;
	CheckNtpSignal:=FALSE;
	RETURN;
END_IF	

// Check NTP is synchronized
IF (NOT i_exNtpSynchronized) THEN
	stat.signal.qos := E_TIME_SIGNAL_QOS.NOT_VALID;
	stat.sErrorMsg := GetErrorText(E_TIME_ERROR.NTP_NOT_SYNCHRONIZED);
END_IF	

// Check time delivered by NTP is not zero. This variable
// shall be mapped to the TcNtpExternalTimeProvider
IF (i_exNtpExtTime = 0) THEN
	stat.signal.qos := E_TIME_SIGNAL_QOS.NOT_VALID;
	stat.sErrorMsg := GetErrorText(E_TIME_ERROR.INT_EXT_NOT_MAPPED);
	CheckNtpSignal:=FALSE;
	RETURN;
END_IF


CheckNtpSignal := TRUE;
END_METHOD

METHOD CheckPtpSignal : BOOL
VAR_INPUT
END_VAR
stat.signal.status :=  E_TIME_SIGNAL_STATUS.CONNECTED;
stat.signal.qos := E_TIME_SIGNAL_QOS.VALID;


// Check external signal. This variable must be mapped to the EL6688 terminal.
IF (i_extDevNotConnected) THEN
	stat.signal.status :=  E_TIME_SIGNAL_STATUS.NOT_CONNECTED;
	stat.signal.qos := E_TIME_SIGNAL_QOS.NOT_VALID;
	CheckPtpSignal:=FALSE;
	RETURN;
END_IF	

// Check DC times computed by EL6688 are not zero. These variables
// shall be mapped to the EL6688 terminal.	
IF ((i_inTime = 0) OR (i_exTime = 0)) THEN
	stat.signal.qos := E_TIME_SIGNAL_QOS.NOT_VALID;
	stat.sErrorMsg := GetErrorText(E_TIME_ERROR.INT_EXT_NOT_MAPPED);
	CheckPtpSignal:=FALSE;
	RETURN;
END_IF

IF (i_dc2TcOffset = GVL_TimeConstants.C_INVALID)  THEN
	stat.signal.qos := E_TIME_SIGNAL_QOS.NOT_VALID;
	stat.sErrorMsg := GetErrorText(E_TIME_ERROR.DC2TC_OFFSET_NOT_MAPPED);
	CheckPtpSignal:=FALSE;
	RETURN;
END_IF
		
// Check quality of the signal synchronization. If the offset from master is
// greater than one second if it is consider not synchronized.
IF (ABS(fb_CoE.GetOffsetFromMaster()) >= GVL_TimeConstants.C_ONE_SEC) THEN
	stat.signal.qos := E_TIME_SIGNAL_QOS.NOT_SYNCHRONIZED;
	stat.sErrorMsg := GetErrorText(E_TIME_ERROR.PTP_NOT_SYNCHRONIZED);
END_IF

// Check CoE diagnostic parameter from EL6688. Terminal shall be
// in SLAVE state and not LISTENNING.

IF (NOT fb_CoE.IsErrorFree()) THEN
	stat.signal.qos := E_TIME_SIGNAL_QOS.NOT_VALID;
	stat.sErrorMsg := GetErrorText(E_TIME_ERROR.COE_NOT_VALID);
	CheckPtpSignal:=FALSE;
	RETURN;
END_IF
	
IF (fb_CoE.GetPtpState() <> E_COE_PTP_STATE.SLAVE) THEN
	stat.signal.status :=  E_TIME_SIGNAL_STATUS.NOT_CONNECTED;
	stat.signal.qos := E_TIME_SIGNAL_QOS.NOT_VALID;
	stat.sErrorMsg := GetErrorText(E_TIME_ERROR.PTP_WRONG_STATE);
	CheckPtpSignal:=FALSE;
	RETURN;
END_IF

CheckPtpSignal := TRUE;
END_METHOD

METHOD ComputeNtpOffset
VAR_INPUT
END_VAR

VAR
	dcExtNtpTime : LINT;
	dcExtNtpLocalTime : LINT;
	tmp : ULINT;
	nFileTime : T_FILETIME;
	str: STRING;
END_VAR



MEMCPY(ADR(nFileTime), ADR(i_exNtpExtTime), SIZEOF(nFileTime));

dcExtNtpTime := FILETIME_TO_DCTIME64(nFileTime);
MEMCPY(ADR(nFileTime), ADR(i_exNtpSysTime), SIZEOF(nFileTime));
dcExtNtpLocalTime := FILETIME_TO_DCTIME64(nFileTime);
stat.lNtpOffsetTime := dcExtNtpLocalTime - dcExtNtpTime;

stat.lTaiTime := stat.lDcCurrentTime - stat.lNtpOffsetTime + (UINT_TO_LINT(cfg.nLeapSecond) * GVL_TimeConstants.C_ONE_SEC);
stat.sTaiTime := DCTIME64_TO_STRING(LINT_TO_ULINT(stat.lTaiTime));

// Convert TAI time from nanoseconds to microseconds
tmp := LINT_TO_ULINT(stat.lTaiTime)/ 10#1000;

// Add offset wrt Unix Base System
tmp := tmp + GVL_TimeConstants.C_UNIX_OFFSET_MICROSEC;

// Convert offset from microseconds to seconds for the MUDPI protocol
stat.lrTaiUnixTimeinSecs := ULINT_TO_LREAL(tmp) / 1000000.0;


stat.lUtcTime := stat.lDcCurrentTime - stat.lNtpOffsetTime;						
stat.sUtcTime := DCTIME64_TO_STRING(LINT_TO_ULINT(stat.lUtcTime));
q_timeInfo.time_offset := stat.lNtpOffsetTime;
q_timeInfo.leap_second := cfg.nLeapSecond;
END_METHOD

METHOD ComputePtpOffset
VAR_INPUT
END_VAR

VAR
	dc2ExtOffset : LINT;
	taiOffset : LINT;
	tmp : LREAL;
END_VAR

dc2ExtOffset := ULINT_TO_LINT(i_inTime) - ULINT_TO_LINT(i_exTime);

taiOffset := dc2ExtOffset + i_dc2TcOffset;

stat.lPtpOffsetTime := (dc2ExtOffset) + i_dc2TcOffset +
                           (GVL_TimeConstants.C_ONE_SEC *  fb_CoE.GetLeapSecond());

stat.lTaiTime := stat.lDcCurrentTime - taiOffset;
stat.sTaiTime := DCTIME64_TO_STRING(LINT_TO_ULINT(stat.lTaiTime));

// Convert TAI time from nanoseconds to microseconds
tmp := LINT_TO_REAL(stat.lTaiTime)/ 10#1000;

// Add offset wrt Unix Base System
tmp := tmp + ULINT_TO_REAL(GVL_TimeConstants.C_UNIX_OFFSET_MICROSEC);

// Convert offset from microseconds to seconds for the MUDPI protocol
stat.lrTaiUnixTimeinSecs := tmp / 1000000.0;

stat.lUtcTime := stat.lDcCurrentTime - stat.lPtpOffsetTime;							
stat.sUtcTime := DCTIME64_TO_STRING(LINT_TO_ULINT(stat.lUtcTime));
q_timeInfo.time_offset := stat.lPtpOffsetTime;
q_timeInfo.leap_second := fb_CoE.GetLeapSecond();
END_METHOD

METHOD ComputeSimulationOffset
VAR_INPUT
END_VAR

VAR
	lSimOffsetTime:	LINT	:= 0;
	tDcUserTime      : ULINT;
	tmp : ULINT;
END_VAR

// Get the time from the user given time string, e.g.
// cfg.sUserTime = '2019-12-07-07:07:07.380500000'
// tDcUserTime   = 629017627380500000
tDcUserTime  := STRING_TO_DCTIME64(cfg.sUserTime);
// Adjust the offset only if user modified the time string.
IF (stat.tUserTime <> tDcUserTime) THEN
	IF (tDcUserTime = 0) THEN
		stat.sErrorMsg := 'ERROR: format of user datetime is not correct';
		RETURN;
	END_IF
	lSimOffsetTime := (stat.lDcCurrentTime - ULINT_TO_LINT(tDcUserTime));
	stat.lSimOffsetTime := lSimOffsetTime;
	stat.tUserTime := tDcUserTime;
END_IF

stat.lUtcTime := stat.lDcCurrentTime - stat.lSimOffsetTime;
stat.sUtcTime := DCTIME64_TO_STRING(LINT_TO_ULINT(stat.lUtcTime));
stat.lTaiTime := stat.lUtcTime + (GVL_TimeConstants.C_ONE_SEC * cfg.nLeapSecond);
stat.sTaiTime := DCTIME64_TO_STRING(LINT_TO_ULINT(stat.lTaiTime));;
// Convert TAI time from nanoseconds to microseconds
tmp := LINT_TO_ULINT(stat.lTaiTime)/ 10#1000;

// Add offset wrt Unix Base System
tmp := tmp + GVL_TimeConstants.C_UNIX_OFFSET_MICROSEC;

// Convert offset from microseconds to seconds for the MUDPI protocol
stat.lrTaiUnixTimeinSecs := ULINT_TO_LREAL(tmp) / 1000000.0;
q_timeInfo.time_offset := stat.lSimOffsetTime;
q_timeInfo.leap_second := cfg.nLeapSecond;
END_METHOD

METHOD CycleUpdate : BOOL
VAR_INPUT
END_VAR
VAR
	fbGetSystemTime  : GETSYSTEMTIME;
    fileTime         : T_FILETIME;
	tDcCurrentTime	 : LINT;
	tDcUserTime      : ULINT;
    sTime            : STRING;
	bSignalOk        : BOOL := FALSE;
END_VAR
VAR_INST
	{attribute 'OPC.UA.DA' := '0'}
	lSimOffsetTime:	LINT	:= 0;
END_VAR
// Get System Time
fbGetSystemTime(timeLoDW=>fileTime.dwLowDateTime, timeHiDW=>fileTime.dwHighDateTime );
stat.sSystemTime := SYSTEMTIME_TO_STRING( FILETIME_TO_SYSTEMTIME( fileTime ) );

// Get DC Time
tDcCurrentTime	:= ULINT_TO_LINT(F_GetCurDcTaskTime64());
stat.lDcCurrentTime := tDcCurrentTime; 
stat.sDcTime := DCTIME64_TO_STRING(LINT_TO_ULINT(tDcCurrentTime));	(* DC time as STRING *)


IF (cfg.nMode =  E_TIME_MODE.LOCAL) THEN
	// In local mode, time used is the time DC time delivered by TwinCAT.
	SetDefaultMode('');
ELSIF (cfg.nMode =  E_TIME_MODE.UTC_PTP)  THEN
	stat.sErrorMsg := '';
	// Check PTP time signal.
	// This will set:
	//	stat.signal.status
	//	stat.signal.qos
	bSignalOk := CheckPtpSignal();
	IF bSignalOk	THEN
		stat.mode := E_TIME_MODE.UTC_PTP;
		ComputePtpOffset();	
	ELSE
		SetDefaultMode('PTP signal NOT ok');
	END_IF
ELSIF (cfg.nMode =  E_TIME_MODE.UTC_NTP)  THEN
	stat.sErrorMsg := '';
	// Check NTP time signal.
	// This will set:
	//	stat.signal.status
	//	stat.signal.qos
	bSignalOk := CheckNtpSignal();
	IF bSignalOk	THEN
		stat.mode := E_TIME_MODE.UTC_NTP;
		// This call computes:
		//	stat.lUtcTime							
		//	stat.sUtcTime
		//	q_timeInfo.time_offset
		ComputeNtpOffset();	
	ELSE
		SetDefaultMode(GetErrorText(E_TIME_ERROR.NTP_NOT_CONNECTED));
	END_IF
ELSIF  (cfg.nMode =  E_TIME_MODE.SIMULATION ) THEN
	// Uses the simulated time
	stat.mode := E_TIME_MODE.SIMULATION;
	stat.sErrorMsg := '';
	// This call computes:
			//	stat.tUserTime							
			//	stat.sUtcTime
			//	q_timeInfo.time_offset
	ComputeSimulationOffset();	
END_IF

q_timeInfo.time_mode := stat.mode;
END_METHOD

METHOD FB_init : BOOL
VAR_INPUT
	bInitRetains : BOOL; // if TRUE, the retain variables are initialized (warm start / cold start)
	bInCopyCode : BOOL;  // if TRUE, the instance afterwards gets moved into the copy code (online change)
END_VAR
stat.sLibVersion := stLibVersion_ESO_LDC_Timer_Library.sVersion;
stat.sErrorMsg := '';
END_METHOD

METHOD GetErrorText : STRING
VAR_INPUT
	i_errorId: DINT;
END_VAR

VAR
	str:	STRING;
END_VAR

CASE i_errorId OF
	E_TIME_ERROR.OK:						str	:= 'OK';
	E_TIME_ERROR.NO_SIMULATION_MODE:	    str	:= 'ERROR: Time can only be set in simulation mode.';	
	E_TIME_ERROR.INT_EXT_NOT_MAPPED:        str := 'ERROR: Did you forget to map the internal or external EL6688 time stamps?';
	E_TIME_ERROR.DC2TC_OFFSET_NOT_MAPPED:   str := 'ERROR: Did you forget to map the dc2tc_offset?';
	E_TIME_ERROR.COE_NOT_VALID:             str := 'ERROR: Error reading COE parameter';
	E_TIME_ERROR.PTP_WRONG_STATE:           str := 'ERROR: EL6688 is not in SLAVE state';
	E_TIME_ERROR.NTP_NOT_CONNECTED:         str := 'ERROR: NTP not connected. Did you forget to map attributes?';
	E_TIME_ERROR.NTP_NOT_SYNCHRONIZED:      str := 'WARNING: NTP not synchronized';
END_CASE

GetErrorText	:= str;
END_METHOD

METHOD GetMode : E_TIME_MODE
VAR_INPUT
END_VAR
GetMode := stat.mode;
END_METHOD

METHOD GetMudpiTime : LREAL
VAR_INPUT
END_VAR

VAR
END_VAR

GetMudpiTime := stat.lrTaiUnixTimeinSecs;
END_METHOD

METHOD GetSource : E_TIME_SOURCE
VAR_INPUT
END_VAR
GetSource := stat.source;
END_METHOD

METHOD GetTime : ULINT
VAR_INPUT
END_VAR

IF (GetMode() =  E_TIME_MODE.LOCAL) THEN
	GetTime := LINT_TO_ULINT(stat.lDcCurrentTime);
END_IF

IF (GetMode() =  E_TIME_MODE.UTC_PTP) THEN
	GetTime := LINT_TO_ULINT(stat.lDcCurrentTime - stat.lPtpOffsetTime);
END_IF

IF (GetMode() =  E_TIME_MODE.UTC_NTP) THEN
	GetTime := LINT_TO_ULINT(stat.lDcCurrentTime - stat.lNtpOffsetTime);
END_IF

IF (GetMode() =  E_TIME_MODE.SIMULATION) THEN
	GetTime := LINT_TO_ULINT(stat.lDcCurrentTime - stat.lPtpOffsetTime);
END_IF
END_METHOD

METHOD GetUtcTime : ULINT
VAR_INPUT
END_VAR

VAR
END_VAR

GetUtcTime := i_exNtpSysTime;
END_METHOD

METHOD MudpiTimeToDc : ULINT
VAR_INPUT
	mudipiTime: LREAL;
END_VAR

VAR
	tmp: LREAL;
END_VAR

// Convert offset from seconds (MUDPI protocol) to microseconds 
tmp := mudipiTime * 1000000.0;

// Remove offset wrt Unix Base System
tmp := tmp - ULINT_TO_LREAL(GVL_TimeConstants.C_UNIX_OFFSET_MICROSEC);

// Convert offset from microseconds to nanoseconds - DC unit
tmp := tmp * 10#1000;

MudpiTimeToDc := LREAL_TO_ULINT(tmp);
END_METHOD

(*
  This method sends the diagnostic data to the TRS system for long term
  monitoring.
  
  The format of the data follows the specification in document ESO-331947.
  The data is sent via UDP packets using the implementation of the MUDPI
  protocol.
  *)

METHOD PublishPtpDiagnostics : BOOL
VAR_INPUT
END_VAR

VAR
    (* TF6311 realtime driver parameters *)
    {attribute 'TcInitSymbol'}
    oid : OTCID;
    ipUdp : ITcIoUdpProtocol;
    nReceivedPackets : UINT;
    uLastReceivedIP : T_IP_ADDRESS;
    hrInit : HRESULT;
    hrSend : HRESULT; 
    bSuccessfulInitializationOfRealtimeDriver : BOOL := FALSE; // Indication of whether the realtime driver is properly initialized.

    (* Data/contents parameters *)
    MudpiPacket : ESO_MUDPI.FB_MudpiPacket(topicId := 500, componentId := 10);

    (* Transmission/communication parameters *)
    _DestinationIpAddress : UDINT; // Destination address for the data
    _DestinationPort : UINT; // Destination port for the data
    _SourcePort : UINT; // Source port of the data

   
END_VAR
END_METHOD

{attribute 'TcRpcEnable':='1'}
METHOD RPC_GetMode : E_TIME_MODE
VAR_INPUT
END_VAR

RPC_GetMode := GetMode();
END_METHOD

{attribute 'TcRpcEnable':='1'}
METHOD RPC_GetUTC : STRING(255)
VAR_INPUT
END_VAR

VAR
	part1: STRING;
	part2: STRING;
	timeStr: STRING(255);
END_VAR

CASE stat.mode OF
	E_TIME_MODE.LOCAL:
		part2 := ' Mode: LOCAL';
	E_TIME_MODE.UTC:
	    part2 := ' Mode: UTC';
	E_TIME_MODE.SIMULATION:
	    part2 := ' Mode: SIMULATION';
END_CASE

part1 := CONCAT('UTC: ', stat.sUtcTime);
timeStr := CONCAT(part1, part2);
RPC_GetUTC := timeStr;
END_METHOD

{attribute 'TcRpcEnable':='1'}
METHOD RPC_SetMode : DINT
VAR_INPUT
	in_mode : E_TIME_MODE;
END_VAR

RPC_SetMode := SetMode(in_mode);
END_METHOD

{attribute 'TcRpcEnable':='1'}
METHOD RPC_SetTime : DINT

VAR_INPUT
	in_time : STRING(29);
END_VAR

RPC_SetTime := SetTime(in_time);
END_METHOD

METHOD SetDefaultMode
VAR_INPUT
	str: STRING := '';
END_VAR

VAR
	tmp : ULINT;
END_VAR
// Time signal not OK. Go to LOCAL mode.
cfg.nMode := E_TIME_MODE.LOCAL;
cfg.nSource := E_TIME_SOURCE.NONE;
stat.mode := E_TIME_MODE.LOCAL;
stat.signal.qos := E_TIME_SIGNAL_QOS.NOT_VALID;
stat.lUtcTime := stat.lDcCurrentTime;
stat.sUtcTime := stat.sDcTime;
IF (str <> '') THEN
	stat.sErrorMsg := str;
END_IF
stat.lTaiTime := stat.lDcCurrentTime;
stat.sTaiTime := stat.sDcTime;
//stat.lSimOffsetTime := 0;  

// Convert TAI time from nanoseconds to microseconds
tmp := LINT_TO_ULINT(stat.lTaiTime)/ 10#1000;
// Add offset wrt Unix Base System
tmp := tmp + GVL_TimeConstants.C_UNIX_OFFSET_MICROSEC;
// Convert offset from microseconds to seconds for the MUDPI protocol
stat.lrTaiUnixTimeinSecs := ULINT_TO_LREAL(tmp) / 1000000.0;				

q_timeInfo.time_offset := 0;
q_timeInfo.leap_second := 0;
END_METHOD

METHOD SetMode : DINT
VAR_INPUT
	i_mode : E_TIME_MODE;
END_VAR

cfg.nMode := i_mode;

SetMode := GVL_TimeConstants.C_STAT_OK;
END_METHOD

METHOD SetSource : DINT
VAR_INPUT
	i_source : E_TIME_SOURCE;
END_VAR

cfg.nSource := i_source;

SetSource := GVL_TimeConstants.C_STAT_OK;
END_METHOD

METHOD SetTime : DINT;

VAR_INPUT
	in_time : STRING(29);
END_VAR

VAR
	dc_time :ULINT;
END_VAR

IF (cfg.nMode <> E_TIME_MODE.SIMULATION) THEN
	stat.sErrorMsg := GetErrorText(E_TIME_ERROR.NO_SIMULATION_MODE); 
	SetTime := E_TIME_ERROR.NO_SIMULATION_MODE;
	RETURN;
END_IF

cfg.sUserTime := in_time;
dc_time := STRING_TO_DCTIME64(in_time);
cfg.tUserTime := dc_time;
//st_stat.lSimOffsetTime := (st_stat.lDcCurrentTime - ULINT_TO_LINT(dc_time));
//q_timeInfo.time_offset := st_stat.lSimOffsetTime;
SetTime := GVL_TimeConstants.C_STAT_OK;
RETURN;
END_METHOD

END_FUNCTION_BLOCK

// POUs/MAIN
PROGRAM MAIN
VAR
	{attribute 'OPC.UA.DA':='1'}
	time_info:	FB_TIME;
END_VAR

time_info();

END_PROGRAM

// VISUs/Templates/GUI_TEMPLATE_TIME
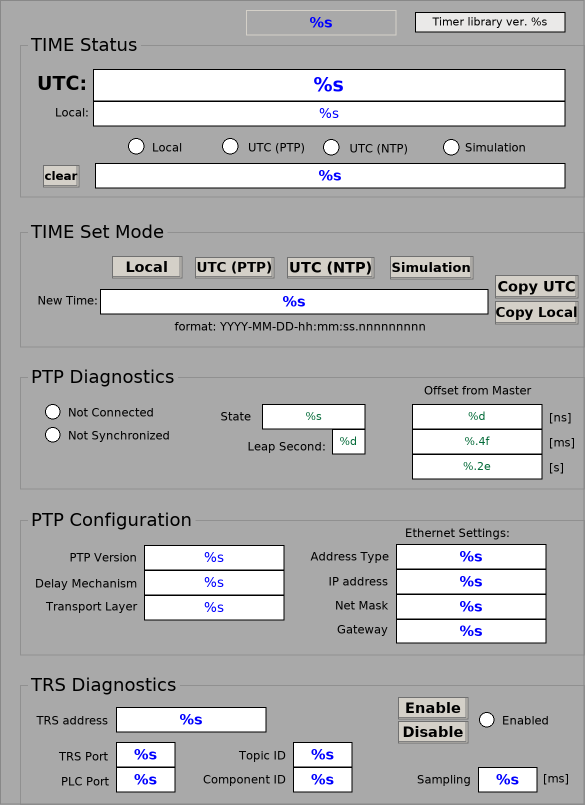
VISUALIZATION GUI_TEMPLATE_TIME  // 585x805
VAR_INPUT
	m_DeviceName : STRING;
END_VAR
VAR_IN_OUT
	m_Instance : FB_TIME;
END_VAR
    GroupBox (20,369 565x120), "PTP Diagnostics"
        Label (391,10 133x23), "Offset from Master"
        Rectangle (242,35 103x25), "%s", text variable: m_Instance.stat.el6688.diagnostics.ptp_state
        Label (192,35 42x25), "State"
        Label (199,65 110x25), "Leap Second:"
        Rectangle (312,60 33x25), "%d", text variable: m_Instance.stat.el6688.diagnostics.leap_second
        Rectangle (392,35 130x25), "%d", text variable: m_Instance.stat.el6688.diagnostics.offset_from_master
        Label (526,35 31x27), "[ns]"
        Rectangle (392,85 130x25), "%.2e", text variable: m_Instance.stat.el6688.diagnostics.offset_from_master_sec
        Label (526,60 31x27), "[ms]"
        Label (526,85 20x27), "[s]"
        Rectangle (392,60 130x25), "%.4f", text variable: m_Instance.stat.el6688.diagnostics.offset_from_master_msec
        Ellipse (25,35 15x15), tooltip "WHITE=Connected RED=Not Connected", colour toggle: (m_Instance.stat.signal.status) = E_TIME_SIGNAL_STATUS.NOT_CONNECTED
        Ellipse (25,58 15x15), tooltip "WHITE=Synchronized RED=Not Synchronized", colour toggle: (m_Instance.stat.signal.qos) = E_TIME_SIGNAL_QOS.NOT_SYNCHRONIZED
        Label (45,31 97x25), "Not Connected"
        Label (45,54 106x25), "Not Synchronized"
    GroupBox (20,37 565x160), "TIME Status"
        Label (23,61 49x29), "Local:"
        Label (113,98 52x25), "Local"
        Rectangle (73,64 472x25), "%s", text variable: m_Instance.stat.sDcTime
        Rectangle (73,32 472x32), "%s", text variable: m_Instance.stat.sUtcTime
        Rectangle (75,126 470x25), "%s", tooltip "Error Message", text variable: m_Instance.stat.sErrorMsg
        Ellipse (108,101 16x16), tooltip "Active time: Local", colour toggle: (m_Instance.stat.mode) = E_TIME_MODE.LOCAL
        Ellipse (202,101 16x16), tooltip "Active time: UTC", colour toggle: (m_Instance.stat.mode = E_TIME_MODE.UTC_PTP)
        Ellipse (423,102 16x16), tooltip "Active time: Simulated", colour toggle: (m_Instance.stat.mode) = E_TIME_MODE.SIMULATION
        Label (430,98 79x25), "Simulation"
        Label (217,98 71x25), "UTC (PTP)"
        Label (321,99 70x25), "UTC (NTP)"
        Ellipse (303,102 16x16), tooltip "Active time: UTC", colour toggle: (m_Instance.stat.mode = E_TIME_MODE.UTC_NTP)
        Button (23,128 36x22), "clear", tooltip "Use local time"
            OnMouseClick: execute { m_Instance.stat.sErrorMsg := ''; }
    GroupBox (20,512 565x143), "PTP Configuration"
        Label (281,80 90x27), "Net Mask"
        Rectangle (376,57 150x25), "%s", text variable: m_Instance.stat.el6688.config.ethernet_settings.ip_address
        Rectangle (376,82 150x25), "%s", text variable: m_Instance.stat.el6688.config.ethernet_settings.subnet_mask
        Label (34,32 86x27), "PTP Version"
        Label (281,105 90x25), "Gateway"
        Rectangle (124,33 140x25), "%s", text variable: m_Instance.stat.el6688.config.ptp_version
        Label (352,7 141x28), "Ethernet Settings:"
        Rectangle (376,107 150x24), "%s", text variable: m_Instance.stat.el6688.config.ethernet_settings.gateway
        Label (7,58 113x27), "Delay Mechanism"
        Rectangle (124,58 140x25), "%s", text variable: m_Instance.stat.el6688.config.delay_mechanism
        Label (10,81 110x27), "Transport Layer"
        Rectangle (376,32 150x25), "%s", text variable: m_Instance.stat.el6688.config.ethernet_settings.address_type
        Rectangle (124,83 140x25), "%s", text variable: m_Instance.stat.el6688.config.transport_layer
        Label (282,30 90x29), "Address Type"
        Label (281,55 90x29), "IP address"
    Label (9,68 81x31), "UTC:"
    Rectangle (246,10 150x25), "%s", text variable: m_DeviceName
    Rectangle (415,12 150x20), "Timer library ver. %s", text variable: m_Instance.stat.sLibVersion
    GroupBox (20,224 565x123), "TIME Set Mode"
        Button (92,32 70x22), "Local", tooltip "Use local time"
            OnMouseClick: execute { m_Instance.cfg.nMode := E_TIME_MODE.LOCAL; }
        Button (175,33 79x21), "UTC (PTP)", tooltip "Use UTC time (source PTP)"
            OnMouseClick: execute { m_Instance.cfg.nMode := E_TIME_MODE.UTC_PTP; }
        Rectangle (80,65 388x25), "%s", tooltip "Time used for Simulation. Press "Copy UTC" or "Copy Local" button to get the time in correct format and then modify it for your needs.", text variable: m_Instance.cfg.sUserTime
            OnMouseDown: write the text variable via Default
        Button (370,32 83x23), "Simulation", tooltip "Use simulated time given under "New Time". NOTE: "New Time" is taken only if the time string has been modified since the last press of the button."
            OnMouseClick: execute { m_Instance.cfg.nMode := E_TIME_MODE.SIMULATION; }
        Label (8,64 73x25), "New Time:"
        Label (139,90 270x25), "format: YYYY-MM-DD-hh:mm:ss.nnnnnnnnn"
        Button (475,51 83x23), "Copy UTC", tooltip "Copy current UTC time to "New Time""
            OnMouseClick: execute { m_Instance.cfg.sUserTime := m_Instance.stat.sUtcTime; }
        Button (267,33 87x21), "UTC (NTP)", tooltip "Use UTC time ((source NTP)"
            OnMouseClick: execute { m_Instance.cfg.nMode := E_TIME_MODE.UTC_NTP; }
    GroupBox (20,677 565x128), "TRS Diagnostics"
        Rectangle (96,65 59x25), "%s", text variable: m_Instance.cfg.diag_report.destination_port
            OnMouseDown: write the text variable via Edit
        Button (378,20 70x22), "Enable", tooltip "Enable Diagnostics"
            OnMouseClick: execute { m_Instance.cfg.diag_report.enabled := TRUE; }
        Button (378,44 70x22), "Disable", tooltip "Disable Diagnostics"
            OnMouseClick: execute { m_Instance.cfg.diag_report.enabled := FALSE; }
        Rectangle (96,90 59x25), "%s", text variable: m_Instance.cfg.diag_report.source_port
            OnMouseDown: write the text variable via Edit
        Label (7,29 84x29), "TRS address"
        Label (479,29 61x29), "Enabled"
        Label (32,65 59x29), "TRS Port"
        Label (23,90 69x29), "PLC Port"
        Label (387,88 67x29), "Sampling"
        Label (521,88 31x27), "[ms]"
        Rectangle (458,90 59x25), "%s", text variable: m_Instance.cfg.diag_report.sampling
            OnMouseDown: write the text variable via Edit
        Ellipse (459,35 15x15), tooltip "WHITE - Disabled GREEN - Enabled", colour toggle: m_Instance.stat.diag_report.enabled
        Rectangle (96,30 150x25), "%s", text variable: m_Instance.cfg.diag_report.address
            OnMouseDown: write the text variable via Edit
        Rectangle (273,65 59x25), "%s", text variable: m_Instance.cfg.diag_report.topic_id
            OnMouseDown: write the text variable via Edit
        Label (210,64 59x29), "Topic ID"
        Label (182,88 87x29), "Component ID"
        Rectangle (273,90 59x25), "%s", text variable: m_Instance.cfg.diag_report.compontent_id
            OnMouseDown: write the text variable via Edit
    Button (495,301 83x23), "Copy Local", tooltip "Copy current Local time to "New Time""
        OnMouseClick: execute { m_Instance.cfg.sUserTime := m_Instance.stat.sDcTime; }
END_VISUALIZATION

// VISUs/GUI_time_info
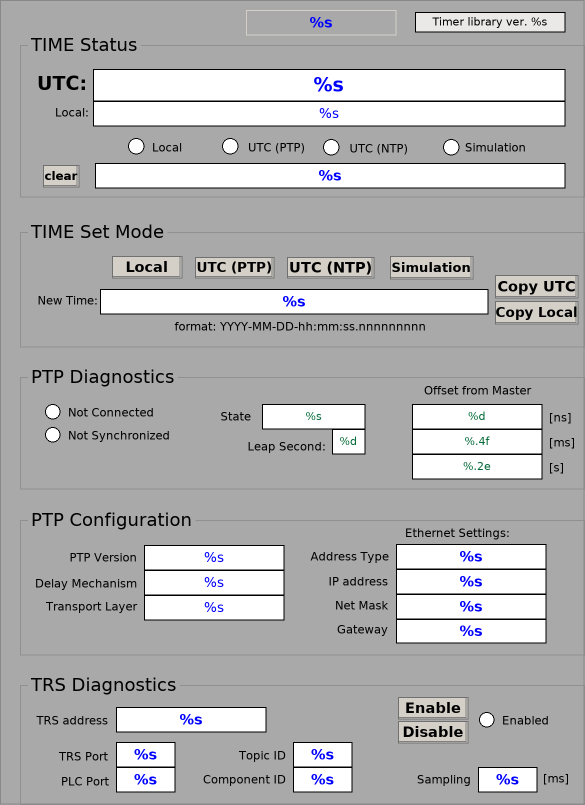
VISUALIZATION GUI_time_info  // 585x805
    Frame (0,0 585x805)
        shows GUI_TEMPLATE_TIME(m_DeviceName := 'time_info', m_Instance := MAIN.time_info)
END_VISUALIZATION
